PROGRAM REMOTE
VAR
	feedback		: RemoteFeedback;	
	control			: RemoteControl;
	
	UdpIO			: UdpClient(3232258620, 50060, 50050, SIZEOF(feedback), ADR(feedback), SIZEOF(control), ADR(control));
	
	enabled			: BOOL := FALSE;
END_VAR

// Control data
IF (control.udp_key <> 81549300) AND enabled THEN
	// COMAU
	COMAU.control.q1 := control.comau.q1;
	COMAU.control.q2 := control.comau.q2;
	COMAU.control.q3 := control.comau.q3;
	COMAU.control.q4 := control.comau.q4;
	COMAU.control.q5 := control.comau.q5;
	COMAU.control.q6 := control.comau.q6;
	COMAU.control.q1_t := control.comau.q1_t;
	COMAU.control.q2_t := control.comau.q2_t;
	COMAU.control.q3_t := control.comau.q3_t;
	COMAU.control.q4_t := control.comau.q4_t;
	COMAU.control.q5_t := control.comau.q5_t;
	COMAU.control.q6_t := control.comau.q6_t;
	COMAU.control.q1_tt := control.comau.q1_tt;
	COMAU.control.q2_tt := control.comau.q2_tt;
	COMAU.control.q3_tt := control.comau.q3_tt;
	COMAU.control.q4_tt := control.comau.q4_tt;
	COMAU.control.q5_tt := control.comau.q5_tt;
	COMAU.control.q6_tt := control.comau.q6_tt;
END_IF

// Time with overflow check
feedback.t := feedback.t + 1.0/1000.0;
IF feedback.t >= 32765.0 THEN
	feedback.t := 0.0;
END_IF

// Feedback data
// EM8000
(*
feedback.em8000.x := EM8000.feedback.Actual_platform_position_surge;
feedback.em8000.y := EM8000.feedback.Actual_platform_position_sway;
feedback.em8000.z := EM8000.feedback.Actual_platform_position_heave;
feedback.em8000.roll := EM8000.feedback.Actual_platform_position_roll;
feedback.em8000.pitch := EM8000.feedback.Actual_platform_position_pitch;
feedback.em8000.yaw	:= EM8000.feedback.Actual_platform_position_yaw;
*)
feedback.em8000.x := SIMULATOR.ship1.x;
feedback.em8000.y := SIMULATOR.ship1.y;
feedback.em8000.z := SIMULATOR.ship1.z;
feedback.em8000.roll := SIMULATOR.ship1.roll;
feedback.em8000.pitch := SIMULATOR.ship1.pitch;
feedback.em8000.yaw	:= SIMULATOR.ship1.yaw;

feedback.em8000.x_t	:= EM8000.feedback.Actual_platform_velocity_surge;
feedback.em8000.y_t	:= EM8000.feedback.Actual_platform_velocity_sway;
feedback.em8000.z_t	:= EM8000.feedback.Actual_platform_velocity_heave;
feedback.em8000.roll_t := EM8000.feedback.Actual_platform_velocity_roll;
feedback.em8000.pitch_t := EM8000.feedback.Actual_platform_velocity_pitch;
feedback.em8000.yaw_t := EM8000.feedback.Actual_platform_velocity_yaw;
feedback.em8000.x_tt := EM8000.feedback.Actual_platform_acceleration_surge;
feedback.em8000.y_tt := EM8000.feedback.Actual_platform_acceleration_sway;
feedback.em8000.z_tt := EM8000.feedback.Actual_platform_acceleration_heave;
feedback.em8000.roll_tt := EM8000.feedback.Actual_platform_acceleration_roll;
feedback.em8000.pitch_tt := EM8000.feedback.Actual_platform_acceleration_pitch;
feedback.em8000.yaw_tt := EM8000.feedback.Actual_platform_acceleration_yaw;
feedback.em8000.L1 := EM8000.feedback.Actual_position_actuator_1;
feedback.em8000.L2 := EM8000.feedback.Actual_position_actuator_2;
feedback.em8000.L3 := EM8000.feedback.Actual_position_actuator_3;
feedback.em8000.L4 := EM8000.feedback.Actual_position_actuator_4;
feedback.em8000.L5 := EM8000.feedback.Actual_position_actuator_5;
feedback.em8000.L6 := EM8000.feedback.Actual_position_actuator_6;

// EM1500
feedback.em1500.x := EM1500.feedback.Actual_platform_position_surge;
feedback.em1500.y := EM1500.feedback.Actual_platform_position_sway;
feedback.em1500.z := EM1500.feedback.Actual_platform_position_heave;
feedback.em1500.roll := EM1500.feedback.Actual_platform_position_roll;
feedback.em1500.pitch := EM1500.feedback.Actual_platform_position_pitch;
feedback.em1500.yaw	:= EM1500.feedback.Actual_platform_position_yaw;
feedback.em1500.x_t	:= EM1500.feedback.Actual_platform_velocity_surge;
feedback.em1500.y_t	:= EM1500.feedback.Actual_platform_velocity_sway;
feedback.em1500.z_t	:= EM1500.feedback.Actual_platform_velocity_heave;
feedback.em1500.roll_t := EM1500.feedback.Actual_platform_velocity_roll;
feedback.em1500.pitch_t := EM1500.feedback.Actual_platform_velocity_pitch;
feedback.em1500.yaw_t := EM1500.feedback.Actual_platform_velocity_yaw;
feedback.em1500.x_tt := EM1500.feedback.Actual_platform_acceleration_surge;
feedback.em1500.y_tt := EM1500.feedback.Actual_platform_acceleration_sway;
feedback.em1500.z_tt := EM1500.feedback.Actual_platform_acceleration_heave;
feedback.em1500.roll_tt := EM1500.feedback.Actual_platform_acceleration_roll;
feedback.em1500.pitch_tt := EM1500.feedback.Actual_platform_acceleration_pitch;
feedback.em1500.yaw_tt := EM1500.feedback.Actual_platform_acceleration_yaw;
feedback.em1500.L1 := EM1500.feedback.Actual_position_actuator_1;
feedback.em1500.L2 := EM1500.feedback.Actual_position_actuator_2;
feedback.em1500.L3 := EM1500.feedback.Actual_position_actuator_3;
feedback.em1500.L4 := EM1500.feedback.Actual_position_actuator_4;
feedback.em1500.L5 := EM1500.feedback.Actual_position_actuator_5;
feedback.em1500.L6 := EM1500.feedback.Actual_position_actuator_6;

// COAMU
feedback.comau.q1 := COMAU.feedback.q1;
feedback.comau.q2 := COMAU.feedback.q2;
feedback.comau.q3 := COMAU.feedback.q3;
feedback.comau.q4 := COMAU.feedback.q4;
feedback.comau.q5 := COMAU.feedback.q5;
feedback.comau.q6 := COMAU.feedback.q6;
feedback.comau.q1_t := COMAU.feedback.q1_t;
feedback.comau.q2_t := COMAU.feedback.q2_t;
feedback.comau.q3_t := COMAU.feedback.q3_t;
feedback.comau.q4_t := COMAU.feedback.q4_t;
feedback.comau.q5_t := COMAU.feedback.q5_t;
feedback.comau.q6_t := COMAU.feedback.q6_t;
feedback.comau.q1_tt := COMAU.feedback.q1_tt;
feedback.comau.q2_tt := COMAU.feedback.q2_tt;
feedback.comau.q3_tt := COMAU.feedback.q3_tt;
feedback.comau.q4_tt := COMAU.feedback.q4_tt;
feedback.comau.q5_tt := COMAU.feedback.q5_tt;
feedback.comau.q6_tt := COMAU.feedback.q6_tt;

// AT960
feedback.at960.x := LREAL_TO_REAL(Main.x);
feedback.at960.y := LREAL_TO_REAL(Main.y);
feedback.at960.z := LREAL_TO_REAL(Main.z);
feedback.at960.q0 := LREAL_TO_REAL(Main.q0);
feedback.at960.q1 := LREAL_TO_REAL(Main.q1);
feedback.at960.q2 := LREAL_TO_REAL(Main.q2);
feedback.at960.q3 := LREAL_TO_REAL(Main.q3);

// MRU1
feedback.mru1.heave := MRU1.feedback.PosMru_D;
feedback.mru1.heave_t := MRU1.feedback.VelMru_D;
feedback.mru1.heave_tt := MRU1.feedback.AccMru_D;
feedback.mru1.turn_rate := MRU1.feedback.AngRate_D;
feedback.mru1.roll := MRU1.feedback.Roll;
feedback.mru1.pitch := MRU1.feedback.Pitch;
feedback.mru1.yaw := MRU1.feedback.Yaw;
feedback.mru1.wx := MRU1.feedback.AngRate_R;
feedback.mru1.wy := MRU1.feedback.AngRate_P;
feedback.mru1.wz := MRU1.feedback.AngRate_Y;
feedback.mru1.wx_t := MRU1.feedback.AngAcc_R;
feedback.mru1.wy_t := MRU1.feedback.AngAcc_P;
feedback.mru1.wz_t := MRU1.feedback.AngAcc_Y;
feedback.mru1.x_t := MRU1.feedback.VelMru_R;
feedback.mru1.y_t := MRU1.feedback.VelMru_P;
feedback.mru1.z_t := MRU1.feedback.VelMru_Y;
feedback.mru1.x_tt := MRU1.feedback.AccMru_R;
feedback.mru1.y_tt := MRU1.feedback.AccMru_P;
feedback.mru1.z_tt := MRU1.feedback.AccMru_Y;

// MRU2
feedback.mru2.heave := MRU2.feedback.PosMru_D;
feedback.mru2.heave_t := MRU2.feedback.VelMru_D;
feedback.mru2.heave_tt := MRU2.feedback.AccMru_D;
feedback.mru2.turn_rate := MRU2.feedback.AngRate_D;
feedback.mru2.roll := MRU2.feedback.Roll;
feedback.mru2.pitch := MRU2.feedback.Pitch;
feedback.mru2.yaw := MRU2.feedback.Yaw;
feedback.mru2.wx := MRU2.feedback.AngRate_R;
feedback.mru2.wy := MRU2.feedback.AngRate_P;
feedback.mru2.wz := MRU2.feedback.AngRate_Y;
feedback.mru2.wx_t := MRU2.feedback.AngAcc_R;
feedback.mru2.wy_t := MRU2.feedback.AngAcc_P;
feedback.mru2.wz_t := MRU2.feedback.AngAcc_Y;
feedback.mru2.x_t := MRU2.feedback.VelMru_R;
feedback.mru2.y_t := MRU2.feedback.VelMru_P;
feedback.mru2.z_t := MRU2.feedback.VelMru_Y;
feedback.mru2.x_tt := MRU2.feedback.AccMru_R;
feedback.mru2.y_tt := MRU2.feedback.AccMru_P;
feedback.mru2.z_tt := MRU2.feedback.AccMru_Y;

UdpIO();

END_PROGRAM

(* stored: Version 1.1.0.1, ProductVersion 3.1.4020.12
   POU REMOTE: Id {4e291570-ebe0-4ba9-b795-df8674c1b54e}, SpecialFunc None *)
